(* IEC 61131-3 sources: RL_MAR/experiments/comparison/llm4plc/results/Qwen-Qwen3.5-9B_20260506_150728/20260506_170441, 1 file *)

(* ---- generated_code_iteration_0.st ---- *)
START_ST
FUNCTION_BLOCK FB_SimpleRepeat
VAR_INPUT
    INPUT_VAR1 : INT := 2;
    INPUT_COUNTER : INT := 4;
END_VAR

VAR_OUTPUT
    OUTPUT_VAR1 : INT;
END_VAR

VAR
    state : INT;
    COUNTER : INT;
    OUTPUT_VAR1_LOCAL : INT;
END_VAR

END_FUNCTION_BLOCK

START_PLAN
0. DECLARE THE NEEDED STATES
STATE 0: INITIALIZE (Set COUNTER to INPUT_COUNTER, set OUTPUT_VAR1 to INPUT_VAR1)
STATE 1: REPEAT_MULTIPLY (Check if COUNTER > 0. If yes, multiply OUTPUT_VAR1 by 2 and decrement COUNTER. If no, transition to STATE 2)
STATE 2: FINALIZE (Assign final OUTPUT_VAR1 to the output variable and reset internal state if needed for next execution)

1. LIST THE OUTPUT VALUES FOR EACH STATE
STATE 0: OUTPUT_VAR1 = INPUT_VAR1, COUNTER = INPUT_COUNTER
STATE 1: OUTPUT_VAR1 = OUTPUT_VAR1 * 2, COUNTER = COUNTER - 1 (Only if COUNTER > 0)
STATE 2: OUTPUT_VAR1 (Final Value) = OUTPUT_VAR1, COUNTER = 0

2. LIST THE TRANSITIONS BETWEEN STATES
STATE 0 -> STATE 1: Always (On first scan or when COUNTER is reset)
STATE 1 -> STATE 2: If COUNTER = 0
STATE 2 -> STATE 0: Always (On next scan to restart or hold final value)

3. DECLARE THE NEEDED VARIABLES
state: INT; // THE STATE VARIABLE (0, 1, 2)
COUNTER : INT; // LOCAL COPY OF INPUT_COUNTER TO DECREMENT
OUTPUT_VAR1_LOCAL : INT; // LOCAL COPY OF INPUT_VAR1 TO MODIFY
END_PLAN
END_ST
